SUBAPPLICATION Uebung_020c4 (* DigitalInput_I1 auf DigitalOutput_Q1; E_TON Einschaltverzögert; Zeit eingeben und speichern, INI *)
  (* Standard: 61499-2; Description: Copyright (c) 2023 Meisterschulen am Ostbahnhof This program and the accompanying materials are made available under the terms of the Eclipse Public License 2.0 which is available at https://www.eclipse.org/legal/epl-2.0/ SPDX-License-Identifier: EPL-2.0 *)
  (* Version 1.0, 2023-10-23, Franz Höpfinger, Meisterschulen am Ostbahnhof, initial API and implementation and/or initial documentation *)
  PACKAGE Uebungen;
  IMPORT Uebungen::const::NVS::NVS_Keys::KEY_I1_STORE;
  IMPORT Uebungen::const::UT::DefaultPool::InputNumber_I1;
  IMPORT logiBUS::io::DI::logiBUS_DI::Input_I1;
  IMPORT logiBUS::io::DQ::logiBUS_DO::Output_Q1;
  IMPORT Uebungen::const::NVS::NVS_Keys::SECTION_I1_STORE;
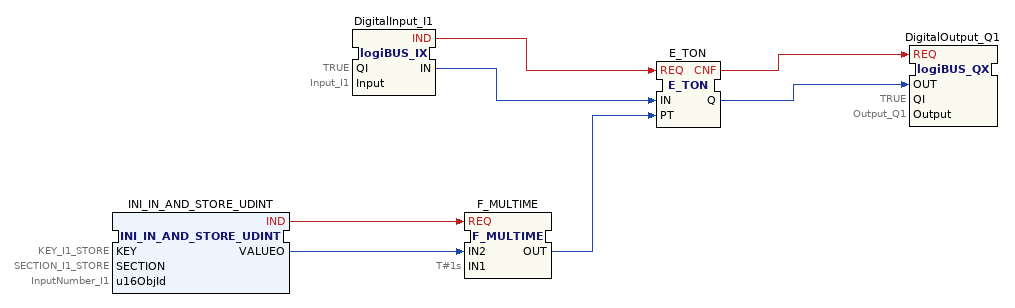
  FBS
    DigitalOutput_Q1 : logiBUS::io::DQ::logiBUS_QX(QI := TRUE, Output := Output_Q1);
    DigitalInput_I1 : logiBUS::io::DI::logiBUS_IX(QI := TRUE, Input := Input_I1);
    E_TON : iec61499::events::timers::E_TON;
    F_MULTIME : iec61131::arithmetic::F_MULTIME(IN1 := T#1s);
  END_FBS
  SUBAPPS
    INI_IN_AND_STORE_UDINT : MyLib::sys::INI_IN_AND_STORE_UDINT(KEY := KEY_I1_STORE, SECTION := SECTION_I1_STORE, u16ObjId := InputNumber_I1);
  END_SUBAPPS
  EVENT_CONNECTIONS
    DigitalInput_I1.IND TO E_TON.REQ;
    E_TON.CNF TO DigitalOutput_Q1.REQ;
    INI_IN_AND_STORE_UDINT.IND TO F_MULTIME.REQ;
  END_CONNECTIONS
  DATA_CONNECTIONS
    DigitalInput_I1.IN TO E_TON.IN;
    E_TON.Q TO DigitalOutput_Q1.OUT;
    F_MULTIME.OUT TO E_TON.PT;
    INI_IN_AND_STORE_UDINT.VALUEO TO F_MULTIME.IN2;
  END_CONNECTIONS
END_SUBAPPLICATION
